// TIA Portal V20 export
DATA_BLOCK "DB81-OPIN"   // DB81
{ S7_Optimized_Access := 'FALSE' }
// stored: AutoNumber false
   VAR
      P001 : Bool;   // P001-T1A - Selectie Mod Operare Manual
      P002 : Bool;   // P002-T1A - Selectie Mod Operare Automat
      P003 : Bool;   // P003-T1A - Ciclu Automat - Cmd. Start
      P004 : Bool;   // P004-Invertere Auxiliare - Reset
      P005 : Bool;   // P005-T1A - Control Pupitru Cabina
      P006 : Bool;   // P006-T1A - Blocare Incarcare
      P007 : Bool;   // P007-T1A - CaleRole - Cmd. Inainte
      P008 : Bool;   // P008-T1A - CaleRole - Cmd. Inapoi
      P009 : Bool;   // P009-T1A - Opritor - Cmd. Inainte
      P010 : Bool;   // P010-T1A - Opritor - Cmd. Inapoi
      P011 : Bool;   // P011-T1A - Lant (transport) - Cmd. Inainte
      P012 : Bool;   // P012-T1A - Lant (transport) - Cmd. Inapoi
      P013 : Bool;   // P013-T1A - Aruncator - Cmd. Sus
      P014 : Bool;   // P014-T1A - Aruncator - Cmd. Jos
      P015 : Bool;   // P015-T1A - Control Pupitru Local
      P016 : Bool;   // P016-T1C - Control Pupitru Cabina
      P017 : Bool;   // P017-T1C - Selectie Mod Operare Manual
      P018 : Bool;   // P018-T1C - Selectie Mod Operare Automat
      P019 : Bool;   // P019-T1C - Ciclu Automat - Cmd. Start
      P020 : Bool;   // P020-T1C - CaleRole - Cmd. Inainte
      P021 : Bool;   // P021-T1C - CaleRole - Cmd. Inapoi
      P022 : Bool;   // P022-T1C - Opritor - Cmd. Inainte
      P023 : Bool;   // P023-T1C - Opritor - Cmd. Inapoi
      P024 : Bool;   // P024-T1C - Lant (transport) - Cmd. Inainte
      P025 : Bool;   // P025-T1C - Lant (transport) - Cmd. Inapoi
      P026 : Bool;   // P026-T1C - Aruncator - Cmd. Sus
      P027 : Bool;   // P027-T1C - Aruncator - Cmd. Jos
      P028 : Bool;   // P028-T1C - Blocare Incarcare
      P029 : Bool;   // P029-T1C - Control Pupitru Local
      P030 : Bool;   // P030-T4 - Selectie Mod Operare Manual
      P031 : Bool;   // P031-T4 - Selectie Mod Operare Automat
      P032 : Bool;   // P032-T4 - Ciclu Automat - Cmd. Start
      P033 : Bool;   // P033-T4 - CaleRole 1 - Cmd. Inainte
      P034 : Bool;   // P034-T4 - CaleRole 1 - Cmd. Inapoi
      P035 : Bool;   // P035-T4 - CaleRole 2 - Cmd. Inainte
      P036 : Bool;   // P036-T4 - CaleRole 2 - Cmd. Inapoi
      P037 : Bool;   // P037-T4 - Lant (rostogolire) - Cmd. Inainte
      P038 : Bool;   // P038-T4 - Lant (rostogolire) - Cmd. Inapoi
      P039 : Bool;   // P039-T4 - Lant (transport) - Cmd. Inainte
      P040 : Bool;   // P040-T4 - Lant (transport) - Cmd. Inapoi
      P041 : Bool;   // P041-T4 - Aruncator - Cmd. Sus
      P042 : Bool;   // P042-T4 - Aruncator - Cmd. Jos
      P043 : Bool;   // P043-T4 - Excentric - Cmd. Inainte
      P044 : Bool;   // P044-T4 - Blocare Rotire Excentric
      P045 : Bool;   // P045-T4 - Excentric - Cmd. Pas
      P046 : Bool;   // P046-T4 - Blocare Descarcare
      P047 : Bool;   // P047-T4 - Excentric - Cmd. Inapoi
      P048 : Bool;   // P048-T1E - Selectie Mod Operare Manual
      P049 : Bool;   // P049-T1E - Selectie Mod Operare Automat
      P050 : Bool;   // P050-T1E - Ciclu Automat - Cmd. Start
      P051 : Bool;   // P051-T1E - CaleRole - Cmd. Inainte
      P052 : Bool;   // P052-T1E - CaleRole - Cmd. Inapoi
      P053 : Bool;   // P053-T1E - Aruncator - Cmd. Sus
      P054 : Bool;   // P054-T1E - Aruncator - Cmd. Jos
      P055 : Bool;   // P055-T1E - Lant Colector - Cmd. Sus
      P056 : Bool;   // P056-T1E - Lant Colector - Cmd. Jos
      P057 : Bool;   // P057-T4 - Lant (rostogolire) - Cmd. Stop
      P058 : Bool;   // P058-T5 - Selectie Mod Operare Manual
      P059 : Bool;   // P059-T5 - Selectie Mod Operare Automat
      P060 : Bool;   // P060-T5 - Ciclu Automat - Cmd. Start
      P061 : Bool;   // P061-T5 - CaleRole - Cmd. Inainte
      P062 : Bool;   // P062-T5 - CaleRole - Cmd. Inapoi
      P063 : Bool;   // P063-T5 - Lant (rostogolire) - Cmd. Inainte
      P064 : Bool;   // P064-T5 - Lant (rostogolire) - Cmd. Inapoi
      P065 : Bool;   // P065-T5 - Lant (transport) - Cmd. Inainte
      P066 : Bool;   // P066-T5 - Lant (transport) - Cmd. Inapoi
      P067 : Bool;   // P067-T5 - Aruncator - Cmd. Sus
      P068 : Bool;   // P068-T5 - Aruncator - Cmd. Jos
      P069 : Bool;   // P069-T5 - Excentric - Cmd. Inainte
      P070 : Bool;   // P070-T5 - Blocare Descarcare
      P071 : Bool;   // P071-T5 - Excentric - Cmd. Pas
      P072 : Bool;   // P072-T5 - Excentric - Cmd. Inapoi
      P073 : Bool;   // P073-T6 - Selectie Mod Operare Manual
      P074 : Bool;   // P074-T6 - Selectie Mod Operare Automat
      P075 : Bool;   // P075-T6 - Ciclu Automat - Cmd. Start
      P076 : Bool;   // P076-T6 - CaleRole - Cmd. Inainte
      P077 : Bool;   // P077-T6 - CaleRole - Cmd. Inapoi
      P078 : Bool;   // P078-T6 - Lant (rostogolire) - Cmd. Inainte
      P079 : Bool;   // P079-T6 - Lant (rostogolire) - Cmd. Inapoi
      P080 : Bool;   // P080-T6 - Lant (transport) - Cmd. Inainte
      P081 : Bool;   // P081-T6 - Lant (transport) - Cmd. Inapoi
      P082 : Bool;   // P082-T6 - Aruncator - Cmd. Sus
      P083 : Bool;   // P083-T6 - Aruncator - Cmd. Jos
      P084 : Bool;   // P084-T6 - Excentric - Cmd. Inainte
      P085 : Bool;   // P085-T6 - Blocare Rotire Excentric
      P086 : Bool;   // P086-T6 - Excentric - Cmd. Pas
      P087 : Bool;   // P087-T6 - Blocare Descarcare
      P088 : Bool;   // P088-T1D - Blocare Incarcare
      P089 : Bool;   // P089-T1D - Selectie Mod Operare Manual
      P090 : Bool;   // P090-T1D - Selectie Mod Operare Automat
      P091 : Bool;   // P091-T1D - Ciclu Automat - Cmd. Start
      P092 : Bool;   // P092-T1D - CaleRole - Cmd. Inainte
      P093 : Bool;   // P093-T1D - CaleRoel - Cmd. Inapoi
      P094 : Bool;   // P094-T1D - Opritor - Cmd. Inainte
      P095 : Bool;   // P095-T1D - Opritor - Cmd. Inapoi
      P096 : Bool;   // P096-T1E - Opritor - Cmd. Inainte
      P097 : Bool;   // P097-T1E - Opritor - Cmd. Inapoi
      P098 : Bool;   // P098-T1D - Aruncator - Cmd. Sus
      P099 : Bool;   // P099-T1D - Aruncator - Cmd. Jos
      P100 : Bool;   // P100-T6 - Excentric - Cmd. Inapoi
      P101 : Bool;   // P101-T7 - Selectie Mod Operare Manual
      P102 : Bool;   // P102-T7 - Selectie Mod Operare Automat
      P103 : Bool;   // P103-T7 - Ciclu Automat - Cmd. Start
      P104 : Bool;   // P104-T7 - CaleRole 1 - Cmd. Inainte
      P105 : Bool;   // P105-T7 - CaleRole 1 - Cmd. Inapoi
      P106 : Bool;   // P106-T7 - CaleRole 2 - Cmd. Inainte
      P107 : Bool;   // P107-T7 - CaleRole 2 - Cmd. Inapoi
      P108 : Bool;   // P108-T7 - Aruncator - Cmd. Sus
      P109 : Bool;   // P109-T7 - Aruncator - Cmd. Jos
      P110 : Bool;   // P110-T7 - Excentric 1 - Cmd. Inainte
      P111 : Bool;   // P111-T7 - Excentric 1 - Cmd. Inapoi
      P112 : Bool;   // P112-T7 - Excentric 1 - Cmd. Pas
      P113 : Bool;   // P113-T7 - Excentric 2 - Cmd. Inainte
      P114 : Bool;   // P114-T7 - Excentric 2 - Cmd. Inapoi
      P115 : Bool;   // P115-T7 - Excentric 2 - Cmd. Pas
      P116 : Bool;   // P116-T7A - Lant (rostogolire) - Cmd. Stop
      P117 : Bool;   // P117-T7ABC - Selectie Pupitru Local pt. T7A, T7B, T7C
      P118 : Bool;   // P118-T7ABC - Selectie Pupitru Cabina pt. T7A, T7B, T7C
      P119 : Bool;   // P119-T7A - Selectie Mod Operare Manual
      P120 : Bool;   // P120-T7A - Selectie Mod Operare Automat
      P121 : Bool;   // P121-T7A - Ciclu Automat - Cmd. Start
      P122 : Bool;   // P122-T7A - CaleRole 1 - Cmd. Inainte
      P123 : Bool;   // P123-T7A - CaleRole 1 - Cmd. Inapoi
      P124 : Bool;   // P124-T7A - CaleRole 2 - Cmd. Inainte
      P125 : Bool;   // P125-T7A - CaleRole 2 - Cmd. Inapoi
      P126 : Bool;   // P126-T7A - Aruncator - Cmd. Sus
      P127 : Bool;   // P127-T7A - Aruncator - Cmd. Jos
      P128 : Bool;   // P128-T7A - Excentric 1 - Cmd. Inainte
      P129 : Bool;   // P129-T7A - Blocare Descarcare
      P130 : Bool;   // P130-T7A - Excentric 1 - Cmd. Pas
      P131 : Bool;   // P131-T7A - Excentric 2 - Cmd. Inainte
      P132 : Bool;   // P132-T7A - Lant (rostogolire) - Cmd. Stop
      P133 : Bool;   // P133-T7A - Excentric 2 - Cmd. Pas
      P134 : Bool;   // P134-T7A - Lant (rostogolire) - Cmd. Inainte
      P135 : Bool;   // P135-T7A - Lant (rostogolire) - Cmd. Inapoi
      P136 : Bool;   // P136-T7A - Lant (transport) - Cmd. Inainte
      P137 : Bool;   // P137-T7A - Lant (transport) - Cmd. Inapoi
      P138 : Bool;   // P138-T7A - Excentric 1 - Cmd. Inapoi
      P139 : Bool;   // P139-T7A - Excentric 2 - Cmd. Inapoi
      P140 : Bool;   // P140-T1A - Lant - Mod Operare Pas
      P141 : Bool;   // P141-T1A - Lant - Mod Operare Continuu
      P142 : Bool;   // P142-T7B - Selectie Mod Operare Manual
      P143 : Bool;   // P143-T7B - Selectie Mod Operare Automat
      P144 : Bool;   // P144-T7B - Ciclu Automat - Cmd. Start
      P145 : Bool;   // P145-T7B - CaleRole - Cmd. Inainte
      P146 : Bool;   // P146-T7B - CaleRole - Cmd. Inapoi
      P147 : Bool;   // P147-T7B - Aruncator 1 - Cmd. Sus
      P148 : Bool;   // P148-T7B - Aruncator 1 - Cmd. Jos
      P149 : Bool;   // P149-T7B - Aruncator 2 - Cmd. Sus
      P150 : Bool;   // P150-T7B - Aruncator 2 - Cmd. Jos
      P151 : Bool;   // P151-T7B - Lant (rostogolire) - Cmd. Inainte
      P152 : Bool;   // P152-T7B - Lant (rostogolire) - Cmd. Inapoi
      P153 : Bool;   // P153-T7B - Lant (transport) - Cmd. Inainte
      P154 : Bool;   // P154-T7B - Lant (transport) - Cmd. Inapoi
      P155 : Bool;   // P155-T7B - Lant Colector - Cmd. Sus
      P156 : Bool;   // P156-T7B - Lant Colector - Cmd. Jos
      P157 : Bool;   // P157- Oprire Sirena Alarma Critica
      P158 : Bool;   // P158-T7C - Selectie Mod Operare Manual
      P159 : Bool;   // P159-T7C - Selectie Mod Operare Automat
      P160 : Bool;   // P160-T7C - Ciclu Automat - Cmd. Start
      P161 : Bool;   // P161-T7C - CaleRole - Cmd. Inainte
      P162 : Bool;   // P162-T7C - CaleRole - Cmd. Inapoi
      P163 : Bool;   // P163-T7C - Aruncator - Cmd. Sus
      P164 : Bool;   // P164-T7C - Aruncator - Cmd. Jos
      P165 : Bool;   // P165-T7C - Lant Colector - Cmd. Sus
      P166 : Bool;   // P166-T7C - Lant Colector - Cmd. Jos
      P167 : Bool;   // P167-T7C - Opritor Mobil - Cmd. Sus
      P168 : Bool;   // P168-T7C - Opritor Mobil - Cmd. Jos
      P169 : Bool;   // P169-T7C - Activare/Dezactivare Reintrare Teva
      P170 : Bool;   // P170-T1C - Lant - Mod Operare Pas
      P171 : Bool;   // P171-T1C - Lant - Mod Operare Continuu
      P172 : Bool;   // P172-LM4 - Control Pupitru Cabina
      P173 : Bool;   // P173-LM4 - Control Pupitru Local
      P174 : Bool;   // P174-LM5 - Control Pupitru Cabina
      P175 : Bool;   // P175-LM5 - Control Pupitru Local
      P176 : Bool;   // P176-LM6 - Control Pupitru Cabina
      P177 : Bool;   // P177-LM6 - Control Pupitru Local
      P178 : Bool;   // P178-T7C - CaleRole - Cmd. Sus
      P179 : Bool;   // P179-T7C - CaleRole - Cmd. Jos
      P180 : Bool;   // P180-Apa - Selectie Mod Operare Manual
      P181 : Bool;   // P181-Apa - Selectie Mod Operare Automat
      P182 : Bool;   // P182-Apa - Ciclu Automat - Cmd. Start
      P183 : Bool;   // P183-T7C - Debitare Selectie Contraprobe
      P184 : Bool;   // P184-Apa - Selectie Insertie/Dezinsertie Destunderizator
      P185 : Bool;   // P185-Apa - Selectie Insertie/Dezinsertie Cap Calire
      P186 : Bool;   // P186-Apa - Pompa 1 (pompa principala) - Cmd. Start
      P187 : Bool;   // P187-Apa - Pompa 1 (pompa principala) - Cmd.Stop
      P188 : Bool;   // P188-Apa - Pompa 2 (pompa principala) - Cmd. Start
      P189 : Bool;   // P189-Apa - Pompa 2 (pompa principala) - Cmd. Stop
      P190 : Bool;   // P190-Apa - Pompa 3 (pompa principala) - Cmd. Start
      P191 : Bool;   // P191-Apa - Pompa 3 (pompa principala) - Cmd. Stop
      P192 : Bool;   // P192-Apa - Pompa 4 (pompa principala) - Cmd. Start
      P193 : Bool;   // P193-Apa - Pompa 4 (pompa principala) - Cmd. Stop
      P194 : Bool;   // P194-Apa - Pompa 5 (pompa turnuri racire) - Cmd. Start
      P195 : Bool;   // P195-Apa - Pompa 5 (pompa turnuri racire) - Cmd. Stop
      P196 : Bool;   // P196-Apa - Pompa 5R - Cmd. Start
      P197 : Bool;   // P197-Apa - Pompa 5R - Cmd. Stop
      P198 : Bool;   // P198-Apa - Pompa 5 - Selectie
      P199 : Bool;   // P199-Apa - Pompa 5R - Selectie
      P200 : Bool;   // P100-Apa - Pompa 8 (pompa drenaj) - Cmd. Start
      P201 : Bool;   // P201-Apa - Pompa 8 (pompa drenaj) - Cmd. Stop
      P202 : Bool;   // P202-Apa - Pompa 9 (pompa tunder) - Cmd. Start
      P203 : Bool;   // P203-Apa - Pompa 9 (pompa tunder) - Cmd. Stop
      P204 : Bool;   // P204-Apa - Pompa 10 (pompa evacuare canal) - Cmd. Start
      P205 : Bool;   // P205-Apa - Pompa 10 (pompa evacuare canal) - Cmd. Stop
      P206 : Bool;   // P206-Apa - Pompa 11 (pompa evacuare avarie) - Cmd. Start
      P207 : Bool;   // P207-Apa - Pompa 11 (pompa evacuare avarie) - Cmd. Stop
      P208 : Bool;   // P208-Apa - Pompa Rez (1-4) Cmd. Start
      P209 : Bool;   // P209-Apa - pompa Rez (1-4) Cmd. Stop
      P210 : Bool;   // P210-Apa - Transportator Elicoidal TE1 - Cmd. Start
      P211 : Bool;   // P211-Apa - Transportator Elicoidal TE1 - Cmd. Stop
      P212 : Bool;   // P212-Apa - Transportator Elicoidal TE2 - Cmd. Start
      P213 : Bool;   // P213-Apa - Transportator Elicoidal TE2 - Cmd. Stop
      P214 : Bool;
      P215 : Bool;   // P215-Dezactivare buzzer
      P216 : Bool;
      P217 : Bool;   // P217-Apa - Ventilator Turn Racire 1 - Cmd. Stop
      P218 : Bool;
      P219 : Bool;   // P219-Apa - Ventilator Turn Racire 2 - Cmd. Stop
      P220 : Bool;   // P220 - Apa - Pompa 1 (pompa principala) - Btn + (Incrementare Setpoint)
      P221 : Bool;   // P220 - Apa - Pompa 1 (pompa principala) - Btn - (Decrementare Setpoint)
      P222 : Bool;   // P222-Apa - Selectie/Deselectie Pompa 1
      P223 : Bool;   // P223-Apa - Selectie/Deselectie Pompa 2
      P224 : Bool;   // P224-Apa - Selectie/Deselectie Pompa 3
      P225 : Bool;   // P225-Apa - Selectie/Deselectie Pompa 4
      P226 : Bool;   // P226-Apa - Selectie/Deselectie Pompa Rez
      P227 : Bool;
      P228 : Bool;   // P228-Apa - Ventilator Turn Racire 1 - Cmd. Start Turatie Mica
      P229 : Bool;   // P229-Apa - Ventilator Turn Racire 1 - Cmd. Start Turatie Mare
      P230 : Bool;   // P230-Apa - Ventilator Turn Racire 2 - Cmd. Start Turatie Mica
      P231 : Bool;   // P231-Apa - Ventilator Turn Racire 2 - Cmd. Start Turatie Mare
      P232 : Bool;   // P232-Apa - Control Pupitru Local
      P233 : Bool;   // P233-Apa - Control Pupitru Cabina
      P234 : Bool;
      P235 : Bool;   // P235-Apa - Y1 - Comanda ON/OFF in Mod Operare Manual
      P236 : Bool;   // P236-Apa - Y2 - Comanda ON/OFF in Mod Operare Manual
      P237 : Bool;   // P237-Apa - Y3 - Comanda ON/OFF in Mod Operare Manual
      P238 : Bool;   // P238-Apa - Deztunderizator - Mod Operare Automat
      P239 : Bool;   // P239-T3 - Deztunderizator - Cmd. Start
      P240 : Bool;   // P240-T3 - Deztunderizator - Cmd. Stop
      P241 : Bool;   // P241-T3 - CaleRole - Cmd. Inainte
      P242 : Bool;   // P242-T3 - CaleRole - Cmd. Inapoi
      P243 : Bool;   // P243-T3 - Cap Calitor 1 - Cmd. Ridicare
      P244 : Bool;   // P244-T3 - Cap Calitor 1 - Cmd. Coborare
      P245 : Bool;   // P245-T3 - Cap Calitor 2 - Cmd. Ridicare
      P246 : Bool;   // P246-T3 - Cap Calitor 2 - Cmd. Coborare
      P247 : Bool;   // P247-T3 - Cap Calitor 3 - Cmd. Ridicare
      P248 : Bool;   // P248-T3 - Cap Calitor 3 - Cmd. Coborare
      P249 : Bool;   // P249-T3 - Grinda - Cmd. Ridicare
      P250 : Bool;   // P250-T3 - Grinda - Cmd. Coborare
      P251 : Bool;   // P251-T3 - Filtru - Cmd. Inainte
      P252 : Bool;   // P252-T3 - Filtru - Cmd. Inapoi
      P253 : Bool;   // P253-T3 - Servovalvola Filtru - Cmd. Start
      P254 : Bool;   // P254-Apa - Deztunderizator - Mod Operare Manual
      P255 : Bool;   // P255-T3 - Servovalvola - Cmd. Start Stropire
      P256 : Bool;   // P256-Apa - Ciclu Automat Deztunderizator - Cmd. Start
      P257 : Bool;   // P257-T7A - Selectie Mod Operare Manual (local)
      P258 : Bool;   // P258-T7A - Selectie Mod Operare Automat (local)
      P259 : Bool;   // P259-T7A - Ciclu Automat - Cmd. Start (local)
      P260 : Bool;   // P260-T7A - CaleRole 1 - Cmd. Inainte (local)
      P261 : Bool;   // P261-T7A - CaleRole 1 - Cmd. Inapoi (local)
      P262 : Bool;   // P262-T7A - CaleRole 2 - Cmd. Inainte (local)
      P263 : Bool;   // P263-T7A - CaleRole 2 - Cmd. Inapoi (local)
      P264 : Bool;   // P264-T7A - Aruncator - Cmd. Sus (local)
      P265 : Bool;   // P265-T7A - Aruncator - Cmd. Jos (local)
      P266 : Bool;   // P266-T7A - Excentric 1 - Cmd. Inainte (local)
      P267 : Bool;   // P267-T7A - Excentric 1 - Cmd. Pas (local)
      P268 : Bool;   // P268-T7A - Excentric 2 - Cmd. Inainte (local)
      P269 : Bool;   // P269-T7A - Excentric 2 - Cmd. Pas (local)
      P270 : Bool;   // P270-T7A - Lant (rostogolire) - Cmd. Inainte (local)
      P271 : Bool;   // P271-T7A - Lant (rostogolire) - Cmd. Inapoi (local)
      P272 : Bool;   // P272-T7A - Lant (transport) - Cmd. Inainte (local)
      P273 : Bool;   // P273-T7A - Lant (transport) - Cmd. Inapoi (local)
      P274 : Bool;   // P274-T7A - Blocare Descarcare (local)
      P275 : Bool;   // P275-T7A - Excentric 1 - Cmd. Inapoi (local)
      P276 : Bool;   // P276-T7A - Excentric 2 - Cmd. Inapoi (local)
      P277 : Bool;   // P277-T4 - Lant - Mod Operare Pas (local)
      P278 : Bool;   // P278-T4 - Lant - Mod Operare Continuu (local)
      P279 : Bool;   // P279-T5 - Lant - Mod Operare Pas (local)
      P280 : Bool;   // P280-T5 - Lant - Mod Operare Continuu (local)
      P281 : Bool;   // P281-T7B - Selectie Mod Operare Manual (local)
      P282 : Bool;   // P282-T7B - Selectie Mod Operare Automat (local)
      P283 : Bool;   // P283-T7B - Ciclu Automat - Cmd. Start (local)
      P284 : Bool;   // P284-T7B - CaleRole - Cmd. Inainte (local)
      P285 : Bool;   // P285-T7B - CaleRole - Cmd. Inapoi (local)
      P286 : Bool;   // P286-T7B - Aruncator 1 - Cmd. Sus (local)
      P287 : Bool;   // P287-T7B - Aruncator 1 - Cmd. Jos (local)
      P288 : Bool;   // P288-T7B - Aruncator 2 - Cmd. Sus (local)
      P289 : Bool;   // P289-T7B - Aruncator 2 - Cmd. Jos (local)
      P290 : Bool;   // P290-T7B - Lant (rostogolire) - Cmd. Inainte (local)
      P291 : Bool;   // P291-T7B - Lant (rostogolire) - Cmd. Inapoi (local)
      P292 : Bool;   // P292-T7B - Lant (transport) - Cmd. Inainte (local)
      P293 : Bool;   // P293-T7B - Lant (transport) - Cmd. Inapoi (local)
      P294 : Bool;   // P294-T7B - Lant Colector - Cmd. Ridicare (local)
      P295 : Bool;   // P295-T7B - Lant Colector - Cmd. Coborare (local)
      P296 : Bool;   // P296-T7B - Lant - Mod Operare Pas
      P297 : Bool;   // P297-T7B - Lant - Mod Operare Continuu
      P298 : Bool;   // P298-T6 - Lant - Mod Operare Pas
      P299 : Bool;   // P299-T6 - Lant - Mod Operare Continuu
      P300 : Bool;   // P300-T7A - Lant - Mod Operare Pas
      P301 : Bool;   // P301-T7A - Lant - Mod Operare Continuu
      P302 : Bool;   // P302-T4 - Reset Tracking
      P303 : Bool;   // P303-T5 - Reset Tracking
      P304 : Bool;   // P304-T6 - Reset Tracking
      P305 : Bool;   // P305-T7C - Selectie Mod Operare Manual (local)
      P306 : Bool;   // P306-T7C - Selectie Mod Operare Automat (loacal)
      P307 : Bool;   // P307-T7C - Ciclu Automat - Cmd. Start (local)
      P308 : Bool;   // P308-T7C - CaleRole - Cmd. Inainte (local)
      P309 : Bool;   // P309-T7C - CaleRole - Cmd. Inapoi (local)
      P310 : Bool;   // P310-T7C - Aruncator - Cmd. Sus (local)
      P311 : Bool;   // P311-T7C - Aruncator - Cmd. Jos (local)
      P312 : Bool;   // P312-T7C - Lant Colector - Cmd. Ridicare (local)
      P313 : Bool;   // P313-T7C - Lant Colector - Cmd. Coborare (local)
      P314 : Bool;   // P314-T7C - Opritor Mobil - Cmd. Sus (local)
      P315 : Bool;   // P315-T7C - Opritor Mobil - Cmd. Jos (local)
      P316 : Bool;   // P316-T7C - CaleRole - Cmd. Sus (local)
      P317 : Bool;   // P317-T7A - Lant - Mod Operare Pas (local)
      P318 : Bool;   // P318-T7A - Lant - Mod Operare Continuu (local)
      P319 : Bool;   // P319-T7B - Lant - Mod Operare Pas (local)
      P320 : Bool;   // P320-T7B - Lant - Mod Operare Continuu (local)
      P321 : Bool;   // P321-T7C - CaleRole - Cmd. Jos (local)
      P322 : Bool;   // P322-T4 - Aliniere Teava - Cap
      P323 : Bool;   // P323-T4 - Aliniere Teava - Coada
      P324 : Bool;
      P325 : Bool;   // P325-T7AB - Activare/Dezactivare Masina Marcare
      P326 : Bool;   // P326-T7AB - Masina Marcare - Cmd. Ridicare
      P327 : Bool;   // P327-T7AB - Masina Marcare - Cmd. Coborare
      P328 : Bool;   // P328-T7AB - Masina Marcare - Cmd. Start Marcare
      P329 : Bool;   // P329-Apa - Selectie Mod Operare Manual (local)
      P330 : Bool;   // P330-Apa - Selectie Mod Operare Automat (local)
      P331 : Bool;   // P331-Apa - Ciclu Automat - Cmd. Start (local)
      P332 : Bool;
      P333 : Bool;
      P334 : Bool;
      P335 : Bool;   // P335-Apa - Pompa 1 (pompa principala) - Cmd. Start (local)
      P336 : Bool;   // P336-Apa - Pompa 1 (pompa principala) - Cmd. Stop (local)
      P337 : Bool;   // P337-Apa - Pompa 2 (pompa principala) - Cmd. Start (local)
      P338 : Bool;   // P338-Apa - Pompa 2 (pompa principala) - Cmd. Stop (local)
      P339 : Bool;   // P339-Apa - Pompa 3 (pompa principala) - Cmd. Start (local)
      P340 : Bool;   // P340-Apa - Pompa 3 (pompa principala) - Cmd. Stop (local)
      P341 : Bool;   // P341-Apa - Pompa 4 (pompa principala) - Cmd. Start (local)
      P342 : Bool;   // P342-Apa - Pompa 4 (pompa principala) - Cmd. Stop (local)
      P343 : Bool;   // P343-Apa - Pompa 5 (pompa turnuri racire) - Cmd. Start (local)
      P344 : Bool;   // P344-Apa - Pompa 5 (pompa turnuri racire) - Cmd. Stop (local)
      P345 : Bool;   // P345-Apa - Pompa 6 (pompa schimbator caldura) - Cmd. Start (local)
      P346 : Bool;   // P346-Apa - Pompa 6 (pompa schimbator caldura) - Cmd. Stop (local)
      P347 : Bool;   // P347-Apa - Pompa 7 (pompa EtilenGlicol) - Cmd. Start (local)
      P348 : Bool;   // P348-Apa - Pompa 7 (pompa EtilenGlicol) - Cmd. Stop (local)
      P349 : Bool;   // P349-Apa - Pompa 8 (pompa drenaj) - Cmd. Start (local)
      P350 : Bool;   // P350-Apa - Pompa 8 (pompa drenaj) - Cmd. Stop (local)
      P351 : Bool;   // P351-Apa - Pompa 9 (pompa tunder) - Cmd. Start (local)
      P352 : Bool;   // P352-Apa - Pompa 9 (pompa tunder) - Cmd. Stop (local)
      P353 : Bool;   // P353-Apa - Pompa 10 (pompa evacuare canal) - Cmd. Start (local)
      P354 : Bool;   // P354-Apa - Pompa 10 (pompa evacuare canal) - Cmd. Stop (local)
      P355 : Bool;   // P355-Apa - Pompa 11 (pompa evacuare avarie) - Cmd. Start (local)
      P356 : Bool;   // P356-Apa - Pompa 11 (pompa evacuare avarie) - Cmd. Stop (local)
      P357 : Bool;
      P358 : Bool;   // Buton oprire aer racire senzori T4
      P359 : Bool;   // P359-Apa - Transportator Elicoidal TE1 - Cmd. Start (local)
      P360 : Bool;   // P360-Apa - Transportator Elicoidal TE2 - Cmd. Stop (local)
      P361 : Bool;   // P361-Apa - Transportator Elicoidal TE2 - Cmd. Start (local)
      P362 : Bool;   // P362-Apa - Transportator Elicoidal TE2 - Cmd. Stop (local)
      P363 : Bool;   // P363-T7C-Masina Debitare: Masina Debitare Comanda Activare/Dezactivare
      P364 : Bool;   // P364-T7C-Masina Debitare: Opritor Mobil Comanda 'Ridicare'
      P365 : Bool;   // P365-T7C-Masina Debitare: Opritor Mobil Comanda 'Coborare'
      P366 : Bool;   // P366-Apa - Ventilator Turn Racire 1 - Cmd. Stop (local)
      P367 : Bool;
      P368 : Bool;   // P368-Apa - Ventilator Turn Racire 2 - Cmd. Stop (local)
      P369 : Bool;   // P369-T7C-Masina Debitare: Menghina Comanda 'Deschide'
      P370 : Bool;   // P370-T7C-Masina Debitare: Menghina Comanda 'Inchide'
      P371 : Bool;   // P371-Apa - Selectie/Deselectie Pompa 1 (local)
      P372 : Bool;   // P372-Apa - Selectie/Deselectie Pompa 2 (local)
      P373 : Bool;   // P373-Apa - Selectie/Deselectie Pompa 3 (local)
      P374 : Bool;   // P374-Apa - Selectie/Deselectie Pompa 4 (local)
      P375 : Bool;   // P375-T7C-Masina Debitare: Lama Circulara Comanda 'Ridicare'
      P376 : Bool;   // P376-T7C-Masina Debitare: Lama Circulara Comanda 'Coborare'
      P377 : Bool;   // P377-Apa - Ventilator Turn Racire 1 - Cmd. Start Turatie Mica (local)
      P378 : Bool;   // P378-Apa - Ventilator Turn Racire 1 - Cmd. Start Turatie Mare (local)
      P379 : Bool;   // P379-Apa - Ventilator Turn Racire 2 - Cmd. Start Turatie Mica (local)
      P380 : Bool;   // P380-Apa - Ventilator Turn Racire 2 - Cmd. Start Turatie Mare (local)
      P381 : Bool;   // P381-T7C-Masina Debitare: Centrala Hidraulica Comanda 'Start'
      P382 : Bool;   // P382-Apa - Y1 - Comanda ON/OFF in Mod Operare Manual
      P383 : Bool;   // P383-Apa - Y2 - Comanda ON/OFF in Mod Operare Manual
      P384 : Bool;   // P384-Apa - Y3 - Comanda ON/OFF in Mod Operare Manual
      P385 : Bool;   // P385 - Reset Oprire de Urgenta - Zona 1
      P386 : Bool;   // P386 - Reset Oprire de Urgenta - Zona 2
      P387 : Bool;   // P387 - Reset Oprire de Urgenta - Zona 3
      P388 : Bool;   // P388 - Reset Oprire de Urgenta - Zona 4
      P389 : Bool;   // P389 - Reset Oprire de Urgenta - Zona 5
      P390 : Bool;   // P390 - Reset Oprire de Urgenta - Zona 6
      P391 : Bool;   // P391 - Reset Oprire de Urgenta - Zona 7
      P392 : Bool;   // P392 - Reset Oprire de Urgenta - Zona 8
      P393 : Bool;   // P393-T7C-Masina Debitare: Centrala Hidraulica Comanda 'Stop'
      P394 : Bool;   // P394-T7AB - Activare/Dezactivare Masina Marcare (local)
      P395 : Bool;   // P395-T7AB - Masina Marcare - Cmd. Ridicare (local)
      P396 : Bool;   // P396-T7AB - Masina Marcare - Cmd. Coborare (local)
      P397 : Bool;   // P397-T7AB - Masina Marcare - Cmd. Start Marcare (local)
      P398 : Bool;   // P398-T1A - Teava Ident
      P399 : Bool;   // P399-T1C - Teava Ident
      P400 : Bool;   // P400-T1D - Teava Ident
      P401 : Bool;   // P401-Apa - Selectie unitate 100bar pentru Destunderizator
      P402 : Bool;   // P402-Apa - Selectie unitate 180bar pentru Destunderizator
      P403 : Bool;   // P403-Apa - Selectat pompa 9.1
      P404 : Bool;   // P404-Apa - Selectat pompa 9.2
      P405 : Bool;   // P405-Apa - Selectat Start pompe joasa presiune
      P406 : Bool;   // P406-Apa - Selectat Stop pompa joasa presiune
      P407 : Bool;   // P407-Apa - Selectat Start pompa inalta presiune
      P408 : Bool;   // P408-Apa - Selectat Stop pompa inalta presiune
      P409 : Bool;   // P409-Apa - Selectat pompa 9.3
      P410 : Bool;   // Marcare-Comanda sus OP local
      P411 : Bool;   // Marcare-Comanda jos OP local
      P412 : Bool;   // Marcare-Comanda sus OP cabina principala
      P413 : Bool;   // Marcare-Comanda jos OP cabina principala
      P414 : Bool;   // P414-Apa - Selectie unitate 200 bar pentru Destunderizator_PSC
      P415 : Bool;   // P409-Apa - Selectat pompa 9.4
      P416 : Bool;
      RK_FW_KEY : Bool;   // P417- Role Kasto - Cmd. Inainte
      RK_BW_KEY : Bool;   // P418- Role Kasto - Cmd. Inapoi
      RM_UP_KEY : Bool;   // P419- Rola Mobila - Cmd. Sus
      RM_DOWN_KEY : Bool;   // P420- Rola Mobila - Cmd. Jos
      TAMPON_LEFT_KEY : Bool;   // P421- Tampon - Cmd. Stanga
      TAMPON_RIGHT_KEY : Bool;   // P422- Tampon - Cmd. Dreapta
      RK_SEL_MANUAL : Bool;   // P423- Taiere Probe Manual
      RK_SEL_AUTOMAT : Bool;   // P424- Taiere Probe Automat
      RK_START_CICLU : Bool;   // P425- Taiere Probe Start Ciclu
      RK_ResetAvarie : Bool;   // Reset avarie zona Kasto
      RK_ReintroduTeava : Bool;   // Reintrodu teava in sistem
      RK_ResetIDBatch : Bool;   // Buton egalizare batch-uri
      P431 : Bool;
      RK_TaiereCapRefulatactiv : Bool;   // Selectie cap refulat activ
      RK_StartTaiere2 : Bool;   // Buton start a doua taiere
      P432 : Bool;   // Start Ventilator Turn 3
      P433 : Bool;   // Stop Ventilator Turn 3
      P434 : Bool;   // Start Ventilator Turn 4
      P435 : Bool;   // Stop Ventilator Turn 4
      P436 : Bool;   // Comanda Scuturator T1C
      P437 : Bool;   // Comanda Scuturator T1A
      P438 : Bool;   // P438 Apa - Pompa 1 Automat
      P439 : Bool;   // P439 Apa - Pompa 1 Manual
      P440 : Bool;
      OCV_CONV_RST : Bool;   // OCV - Reset Convertizor [Main Cabin]
      OCV_CONV_HOME_MCB : Bool;   // OCV - Home Convertizor [Main Cabin]
      OCV_LED_ON_MCB : Bool;   // OCV - LED On [Main Cabin]
      OCV_LED_OFF_MCB : Bool;   // OCV - LED Off [Main Cabin]
      OCV_CAM_START_MCB : Bool;   // OCV - Start Camera [Main Cabin]
      OCV_MOVE_UP_MCB : Bool;   // OCV - Ridicare [Main Cabin]
      OCV_MOVE_DW_MCB : Bool;   // OCV - Coborare [Main Cabin]
      OCV_CLEAN_CMD_MCB : Bool;   // OCV - Curatare Cap Marcare [Main Cabin]
      OCV_PURGE_CMD_MCB : Bool;   // OCV - Purjare Cap Marcare [Main Cabin]
      OCV_CONV_HOME_LM7 : Bool;   // OCV - Home Convertizor [LM7]
      OCV_LED_ON_LM7 : Bool;   // OCV - LED On [LM7]
      OCV_LED_OFF_LM7 : Bool;   // OCV - LED Off [LM7]
      OCV_CAM_START_LM7 : Bool;   // OCV - Start Camera [LM7]
      OCV_MOVE_UP_LM7 : Bool;   // OCV - Ridicare [LM7]
      OCV_MOVE_DW_LM7 : Bool;   // OCV - Coborare [LM7]
      OCV_CLEAN_CMD_LM7 : Bool;   // OCV - Curatare Cap Marcare [LM7]
      OCV_PURGE_CMD_LM7 : Bool;   // OCV - Purjare Cap Marcare [LM7]
      var_bool : Array[0..70] of Int;
   END_VAR
BEGIN
END_DATA_BLOCK
